fbIbBottleTransferAfterDragAfterSensor		(bIN:=
											P00_PackML.fbPMLAuto.ePMLState = E_PMLState.ePMLState_EXECUTE AND P13_BottleTransferAfterDrag.IbBottleTransferAfterDragAfterSensor													
											,tFilterTimeOn:=T#0MS, tFilterTimeOff:=T#500MS);
fbIbBottleTransferAfterDragSecondFormSensor		(bIN:=
											P00_PackML.fbPMLAuto.ePMLState = E_PMLState.ePMLState_EXECUTE AND P13_BottleTransferAfterDrag.IbBottleTransferAfterDragSecondFormSensor													
											,tFilterTimeOn:=T#35MS, tFilterTimeOff:=T#35MS);
rtfbIbBottleTransferAfterDragSecondFormSensor (CLK:=fbIbBottleTransferAfterDragSecondFormSensor.bOUT,Q=>);
IF rtfbIbBottleTransferAfterDragSecondFormSensor.Q THEN
	rtfbIbBottleTransferAfterDragSecondFormSensorCounter := rtfbIbBottleTransferAfterDragSecondFormSensorCounter + 1;
END_IF
tonrtfbIbBottleTransferAfterDragSecondFormSensorCounter(IN:=	rtfbIbBottleTransferAfterDragSecondFormSensorCounter<2 AND 
																P13_BottleTransferAfterDrag.IbBottleTransferAfterDragFirstFormSensor AND
																P13_BottleTransferAfterDrag.IbBottleTransferAfterDragSecondFormSensor AND
																bFormTransportersAfterScrewerCmdStart
														,PT := T#10S);
IF tonrtfbIbBottleTransferAfterDragSecondFormSensorCounter.Q THEN
	rtfbIbBottleTransferAfterDragSecondFormSensorCounter := 2;
END_IF

tonBottleTransferAfterDrag (IN:= 
								(P00_PackML.fbPMLAuto.ePMLState = E_PMLState.ePMLState_EXECUTE) AND 
								NOT (P00_PackML.fbPMLAuto.ePMLState = E_PMLState.ePMLState_STOPPING) AND
								P13_BottleTransferAfterDrag.fbBottleTransferAfterDrag.eState = E_Station.eReady AND 

								P13_BottleTransferAfterDrag.IbBottleTransferAfterDragFirstFormSensor AND
								rtfbIbBottleTransferAfterDragSecondFormSensorCounter >=2 
								//P13_BottleTransferAfterDrag.IbBottleTransferAfterDragSecondFormSensor,	
							,PT:=T#0MS);
P01_PucksInserter.IbPucksInserterFormGateAfterSensor;// Czujnik za PI						
						
IF tonBottleTransferAfterDrag.Q AND 
	NOT P13_BottleTransferAfterDrag.fbBottleTransferAfterDrag.bCycleDone AND
	NOT fbIbBottleTransferAfterDragAfterSensor.bOUT
THEN
	VIS.bBottleTransferAfterDragRun	:= TRUE;
END_IF

IF P13_BottleTransferAfterDrag.fbBottleTransferAfterDrag.bCycleDone THEN
	VIS.bBottleTransferAfterDragRun	:= FALSE;
	rtfbIbBottleTransferAfterDragSecondFormSensorCounter:= 0;
END_IF
END_ACTION

ACTION aP14_BadBottleConveyor:

(*************TRANSPORTER ODRZUCONYCH BUTELEK****************)
(************Przeniesiono wyzej*****************************)

(*Załączany w programie robota jak jest dorzut butelki i kasowany po 30 sekundach*)
IF bBadBottleConveyorEnable THEN
	;
ELSE
	bBadBottleConveyorStart				:=	FALSE;
	bBadBottleConveyorStartTriggerDelay	:=	FALSE;
END_IF

//Opóznienie załączania transporeta
IF bBadBottleConveyorStartTriggerDelay AND P13_BottleTransfer.fbBottleTransfer.eRunningState = eRejected THEN
	bBadBottleConveyorStartTrigger			:= TRUE;
	bBadBottleConveyorStartTriggerDelay		:=FALSE;
END_IF

//Sterowanie transporterem odrzuconych butelek
rtBadBottleConvoyerStart	(CLK:=	bBadBottleConveyorStartTrigger);
tofBadBottleConveyorStart	(IN:=	rtBadBottleConvoyerStart.Q ,	PT:=T#10S);

IF rtBadBottleConvoyerStart.Q THEN //Uruchamianie na cykl
	bBadBottleConveyorStartTrigger		:=	FALSE;
END_IF
IF NOT tofBadBottleConveyorStart.Q  THEN
	bBadBottleConveyorStart				:=	FALSE;
	bBadBottleConveyorStartTrigger		:=	FALSE;
ELSE
	bBadBottleConveyorStart 			:=	TRUE;	
END_IF
END_ACTION

ACTION aP15_FormTransporters:
(********Transporter przed dozownikami*************)
tofbFormTransportersDispencerSlow			(IN:=bFormTransportersDispencerSlowSpeedPulse, 	PT:=T#60S);
tonbFormTransportersDispencerResetSpeed		(IN:=bFormTransportersDispencerResetSpeed, 		PT:=T#5S);
tonQueBeforeScrewers						(IN:=P10_GripperScrewer.IbGripperScrewersSixthFormCheckFormSensor, PT:=T#1500mS);
tonQueAfterScrewers							(IN:=P11_CapCorrectCheck.IbCapCorrectCheckAfterScrewerFormSensor AND P11_CapCorrectCheck.IbCapCorrectCheckDialAfterScrewerFormSensor, PT:=T#2S);
tonQueAfterPlatin							(IN:=MAIN.IbLidSealerAfterSensor, PT:=T#3S);
tonQueBeforeDispencers						(IN:=MAIN.IbFormCheckFormSensor, PT:=T#2S);
tonDelayedStartAfterDisp					(IN:=NOT P09_CapPuttedCheck.fbIbCapPuttedCheckFormSensor.bOUT, PT:=T#1.5S);
IF GVL.bFormTransportersEnable AND (P00_PackML.fbPMLAuto.ePMLState = E_PMLState.ePMLState_EXECUTE)  THEN
	IF NOT VIS.bDosingTwoPhasesShow  THEN
		bFormTransportersDispencerCmdStart := TRUE;
	ELSIF VIS.bDosingTwoPhasesShow AND	NOT bFormTransportersScrewerStop AND NOT tonQueAfterPlatin.q THEN
		bFormTransportersDispencerCmdStart := TRUE;	
	END_IF
	bFormTransportersDispencerSlowSpeedPulse	:=	FALSE;
	(*Spowalnianie transportera*)	
	IF tofbFormTransportersDispencerSlow.Q AND NOT tonbFormTransportersDispencerResetSpeed.Q THEN
		bFormTransportersDispencerSlowSpeed	:= NOT VIS.bCapPuttedCheckIgnoreErrors; 
	ELSE
		bFormTransportersDispencerSlowSpeed	:= FALSE;
	END_IF
	IF bDosingTwoPhases THEN
		bFormTransportersDispencerSlowSpeed	:= TRUE;
	END_IF	
END_IF
	(*Wydmuch na tym transporterze*)
	QbBlowAfterGripperScrewer :=	bFormTransportersDispencerSlowSpeed;
(********Koniec Transporter przed dozownikami********)
	
(********Transporter za dozownikami*************)
tonbFormTransportersScrewerStop	(IN:=	(P05_Weight.eWeightStationRunningState = E_WeightLiftStationState.eStorageOfForms) AND 
										P05_Weight.fbWeightStation.iFormsCounterWeight1 >=3 AND 
										P05_Weight.fbWeightStation.iFormsCounterWeight2 >=3 AND 
										P05_Weight.fbWeightStation.iFormsCounterWeight3 >=3 AND 
										P05_Weight.fbWeightStation.iFormsCounterWeight4 >=3,
									PT:=T#500MS);
tofFormTransportersScrewerSlowSpeed	(IN:=P00_ReadRFIDCard.bReadedCardCapSorter AND bDosingTwoPhases, PT:=T#2S500MS);

IF 	P10_GripperScrewer.fbGripperScrewersDragStation.eRunningState = E_DragStationState.eEndingOfDrag  OR tonThirdFormCheckFormSensor.q THEN
//IF 	P10_GripperScrewer.fbGripperScrewersDragStation.eRunningState = E_DragStationState.eDraging AND P10_GripperScrewer.QbGripperScrewersDragLeadBefore1Actuator THEN
	bFormTransportersScrewerStop			:= FALSE;
END_IF


IF tonLongDelayAfterStart.Q AND
		eBeforeCapSorterPackageState[4].bFormPresent  AND
		(tonCapSorterFourthFormatSensorAnRegister.Q AND iCapSorterDragFormCounter >= 4)AND 
		MAIN.IbCapSorterBeforeFourthFormCheckFormSensor 
		THEN
			IF 
				NOT (
					(P05_Weight.eWeightStationRunningState = E_WeightLiftStationState.eStorageOfForms) AND 
					P05_Weight.fbWeightStation.iFormsCounterWeight1 =3 AND 
					P05_Weight.fbWeightStation.iFormsCounterWeight2 =3 AND 
					P05_Weight.fbWeightStation.iFormsCounterWeight3 =3 AND 
					P05_Weight.fbWeightStation.iFormsCounterWeight4 =3 
					)
				AND NOT bFormTransportersScrewerStop	
				//?AND NOT bLidFeederEnable
				(*AND NOT bDosingTwoPhases*)
				AND NOT bPhaseChanging
				AND tonDelayAfterStart.Q
				//AND (tonQueAfterScrewers.Q OR tonQueBeforeScrewers.Q)  //vs testy
			THEN
				bFormTransportersScrewerStop				:= 	TRUE;
			END_IF
		//bFormTransportersScrewerStop				:= 	TRUE;
END_IF
tonQueAfterScrewers.Q; tonQueBeforeScrewers.Q;
//IF bFormTransportersEnable AND (P00_PackML.fbPMLAuto.ePMLState = E_PMLState.ePMLState_EXECUTE)THEN //dp
IF bDelayAfterStart AND (*tonDelayAfterStart.Q AND*) bFormTransportersEnable AND (P00_PackML.fbPMLAuto.ePMLState = E_PMLState.ePMLState_EXECUTE OR 
		P00_PackML.fbPMLAuto.ePMLState = E_PMLState.ePMLState_STOPPING) (*AND tonDelayedStartAfterDisp.q co to*) THEN
	bFormTransportersScrewerCmdStart 			:= TRUE;
	tonbCapSorterOrCapSorterDragError.Q; 		//Spowalnianie transportera dla wag
	IF bFormTransportersScrewerStop	(*AND NOT tonbCapSorterOrCapSorterDragError.Q)*) THEN //Zatrzymywanie
		bFormTransportersScrewerCmdStart 		:= FALSE;
		
	END_IF
	//Vasyl na prośbę Karola
	(*IF (VIS.bDosingTwoPhasesShow OR vis.bLidFeederEnableShow) AND	tonQueAfterPlatin.Q OR bFormTransportersScrewerStop AND tonQueBeforeDispencers.q THEN
		bFormTransportersDispencerCmdStart 		:= FALSE;
	END_IF*)
END_IF

(********Transporter za sorterem nasadek*************)
IF bFormTransportersEnable AND (P00_PackML.fbPMLAuto.ePMLState = E_PMLState.ePMLState_EXECUTE)  THEN
	bFormTransportersAfterCapSorterCmdStart := TRUE;
	IF tonQueBeforeScrewers.Q THEN
		bFormTransportersAfterCapSorterCmdStart := FALSE;
	END_IF
END_IF	
	
(********Transporter przed zakręcarkami**************)
IF bFormTransportersEnable AND (P00_PackML.fbPMLAuto.ePMLState = E_PMLState.ePMLState_EXECUTE)  THEN
	bFormTransportersBeforeScrewerCmdStart := TRUE;
END_IF	

(*Wydmuch na tym transporterze*)
fbIbBlowBeforeGripperScrewerSensor		(bIn:=MAIN.IbBlowBeforeGripperScrewerSensor, tFilterTimeon:=T#5MS, tFilterTimeOff:=T#300MS);
fbIbBlowBeforeGripperScrewerSensor2		(bIn:=MAIN.IbBlowBeforeGripperScrewerSensor, tFilterTimeon:=T#100MS, tFilterTimeOff:=T#300MS);
tonBlowBeforeGripperScrewerSensor 		(IN:=MAIN.IbBlowBeforeGripperScrewerSensor, PT:=T#15S);
tpfbIbBlowBeforeGripperScrewerSensor 	(IN:=fbIbBlowBeforeGripperScrewerSensor.bOUT, PT:=T#1S);
QbBlowBeforeGripperScrewer	:=	fbIbBlowBeforeGripperScrewerSensor.bOut AND NOT tonBlowBeforeGripperScrewerSensor.Q;

(*Spowalniacz/szlabanik przed zakrecarkami*)
fbIbGateBeforeGripperScrewerSensor 		(bIn:=IbGateBeforeGripperScrewerSensor, tFilterTimeon:=T#20MS, tFilterTimeOff:=T#0MS);
fb2IbGateBeforeGripperScrewerSensor 	(bIn:=IbGateBeforeGripperScrewerSensor, tFilterTimeon:=T#400MS, tFilterTimeOff:=T#0MS);//bylo 670
ftfbIbGateBeforeGripperScrewerSensor	(CLK:=fbIbGateBeforeGripperScrewerSensor.bOUT,	Q=>);	
IF ftfbIbGateBeforeGripperScrewerSensor.Q THEN
	bGateBeforeGripperScrewer	:= TRUE;
END_IF
tonbGateBeforeGripperScrewer			(IN:=bGateBeforeGripperScrewer, PT:=T#400MS);
IF tonbGateBeforeGripperScrewer.Q THEN
	bGateBeforeGripperScrewer	:= FALSE;
END_IF
toniGateBeforeGripperScrewerCase1 (IN:=	iGateBeforeGripperScrewerCase = 10, PT:=T#4S);
						
CASE iGateBeforeGripperScrewerCase OF
	0:
		QbGateBeforeGripperScrewer 		:=	TRUE;
		iGateBeforeGripperScrewerCase	:=	iGateBeforeGripperScrewerCase	+	10;
	10:
		IF toniGateBeforeGripperScrewerCase1.Q AND NOT P09_CapPuttedCheck.IbCapPuttedCheckFormSensor THEN
			iGateBeforeGripperScrewerCase	:=	iGateBeforeGripperScrewerCase	+	10;
		END_IF
	20:
		QbGateBeforeGripperScrewer		:=	FALSE;
		iGateBeforeGripperScrewerCase	:=	iGateBeforeGripperScrewerCase	+	10;
	30: 
		QbGateBeforeGripperScrewer :=		fb2IbGateBeforeGripperScrewerSensor.bOUt;
END_CASE
	
//Spowalnianie formatek
iFormBeforeScrewers := 		
                       		BOOL_TO_INT(eBeforeScrewers2PackageState[2].bFormPresent)+
                       		BOOL_TO_INT(eBeforeScrewers2PackageState[1].bFormPresent)+
                       		BOOL_TO_INT(eBeforeScrewersPackageState[2].bFormPresent)+
                       		BOOL_TO_INT(eBeforeScrewersPackageState[1].bFormPresent);

tonCapPuttedFormsCheck			(IN:=	P10_GripperScrewer.IbGripperScrewersSixthFormCheckFormSensor,		PT:=T#80MS); //bylo 130
tonThirdFormCheckFormSensor		(IN:=	NOT P10_GripperScrewer.IbGripperScrewersSixthFormCheckFormSensor ,	PT:=T#30MS);
IF // Zatrzymywanie jeżeli
	tonCapPuttedFormsCheck.Q OR 			
	P00_PackML.fbPMLAuto.ePMLState = E_PMLState.ePMLState_STOPPING 	OR	
	NOT tonDelayAfterStart.Q	
THEN
	bFormTransporterSlowerCmdStart := FALSE;
END_IF
IF bDelayAfterStart AND bFormTransportersEnable AND 
	(
		tonThirdFormCheckFormSensor.Q OR 
		(NOT bDelayAfterStartFullRegister AND NOT P09_CapPuttedCheck.IbCapPuttedCheckFormSensor) OR
		(bDelayAfterStartFullRegister AND iFormBeforeScrewers=2) //do usuniecia
	)
	AND
	NOT (P00_PackML.fbPMLAuto.ePMLState = E_PMLState.ePMLState_STOPPING) 
	THEN 
		bFormTransporterSlowerCmdStart := TRUE;
END_IF

(********Transporter za zakręcarkami**************)
IF bFormTransportersEnable AND (P00_PackML.fbPMLAuto.ePMLState = E_PMLState.ePMLState_EXECUTE)  THEN
	bFormTransportersAfterScrewerCmdStart := TRUE;
END_IF
END_ACTION

ACTION aP16_LabelMachines:
(***********P16_LabelMachines**************)
(******************************************)
IF bLabelMachineEnable THEN
	bLabelMachineCmdStart := TRUE;
ELSE
	bLabelMachineCmdStart := FALSE;	
END_IF
(******************************************)
(******************************************)
END_ACTION

ACTION aP17_TurnTables:
(************P17_TurnTables****************)
(******************************************)

IF bExitTurnTableEnable AND bDelayAfterStart THEN
	bExitTurnTableCmdStart := TRUE;
ELSIF bDelayAfterStart THEN
	;//bExitTurnTableCmdStart := FALSE;
END_IF
(******************************************)
(******************************************)
IF bExitConveyorEnable AND bDelayAfterStart THEN
	bExitConveyorCmdStart := TRUE;
ELSE
	;//bExitConveyorCmdStart := FALSE;
END_IF
(******************************************)
(******************************************)


(*********************************************************)
(*********Szlaban na transporterze odbiorczym*************)
//Jeżeli stół pracuje 
bExitConveyorCmdStart;
//To ruszaj szlabanem
bExitConveyorGateRun;
//Czujnik z szlabanem
P17_TurnTables.IbExitConveyorGateAfterSensor;
P17_TurnTables.IbExitConveyorGateAfterSensor2;
IF bExitConveyorCmdStart THEN
	fbIbExitConveyorGateAfterSensor		(bIN:=P17_TurnTables.IbExitConveyorGateAfterSensor,	tFilterTimeOn:=T#10MS,	tFilterTimeOff:=T#10MS);
	fbIbExitConveyorGateAfterSensor2	(bIN:=P17_TurnTables.IbExitConveyorGateAfterSensor2,tFilterTimeOn:=T#1S800MS,	tFilterTimeOff:=T#1S800MS);
	tonbExitConveyorGateRun				(IN:=bExitConveyorGateRun AND NOT fbIbExitConveyorGateAfterSensor.bOUT, 	PT:=T#300MS);
	
	bExitConveyorGateRun S= fbIbExitConveyorGateAfterSensor.bOut;	
	bExitConveyorGateRun R= tonbExitConveyorGateRun.Q;	
	
	IF fbIbExitConveyorGateAfterSensor2.bOut AND bExitConveyorGateRun THEN
		bExitConveyorGateRunTemp := TRUE;
	ELSIF NOT fbIbExitConveyorGateAfterSensor2.bOut THEN
		bExitConveyorGateRunTemp := FALSE;	
	END_IF
	IF bExitConveyorGateRunTemp THEN
		bExitConveyorGateRun	:=	TRUE;
	END_IF
END_IF
(*********************************************************)
(*********************************************************)
	fbIbExitConveyorGateAfterSensor3		(bIN:=P17_TurnTables.IbExitConveyorGateAfterSensor,	tFilterTimeOn:=T#10MS,	tFilterTimeOff:=T#12S);

IF tonNotExecute.Q AND NOT fbIbExitConveyorGateAfterSensor3.bOut THEN
	bExitTurnTableCmdStart := FALSE;
	bExitConveyorCmdStart := FALSE;
END_IF
END_ACTION

END_PROGRAM

(* stored: Version 1.1.0.1, ProductVersion 3.1.4026.13, FileIdentifier 411a00112639a9e7228e2dd2d6e06ed5d9c97a99, FileSignature 68d56f6f7cd023b1b7825046622d1bf8a0b812843790b8bb4421e9821bde7a660f56d9956663ebebe51dd14dbbf8236e075714483451083181fa8ec4dce18396552c98323adbd34d97d4a2183e173e6a79f00ccb83a6e16e8aa8d04c780698a18ddc75a4fdb53c6e0a5ad36b78cb566d6a015d5d488b0f36d33e108bc6e3947adc481485b9a785ae4955bba34f0f1973acdd1e36ad2dc3e1a0f49b4145bd6d87dcf949c93894586451675c2a70766f69423c8f864f2bd740daf309413cd2660d30a041a2064fbf69f03032e63452ecfc9f4f022dbc58b6cc8660d268e867e61278df3a041a7dc567f471a15f51f76fbc6f01ffd4ca64c70a460cc0ac4c56d873
   POU P00_PackML: Id {bb851725-25aa-4e37-a964-31b2adf51159}, SpecialFunc None
   Folder CycleLogic: Id {06cd4f29-1d4a-4562-a5b5-d65a5d63923d}
   Folder Homing: Id {cd69f01d-dff3-44b8-b479-c86f6f37d13a}
   Folder Others: Id {4eaa7fda-3f18-47f1-b364-12a902042f69}
   Folder PML: Id {0da3c268-e19f-41cb-aa11-c303f93e5e7c}
   Folder PMLCommonStates: Id {650a41a5-55ef-4702-bbaa-88ebcf63e664}
   Action ACT_Aborted: Id {58aa837e-c8fc-4c28-9ce0-4a427a6cab20}
   Action ACT_Aborting: Id {6a678a84-5a61-4250-a4be-abf00b56123e}
   Action ACT_AntyError: Id {c7865532-fee1-4504-9555-bab70b080968}
   Action ACT_CapSorterBottleSorterAutoStart: Id {c3fb2df5-496e-4d6e-b52b-194c6aba5684}
   Action ACT_Clearing: Id {4fb303d6-b538-45f5-9c59-d20965484409}
   Action ACT_CycleLogic: Id {3da44b98-718e-4e63-9d16-900d089a9e0c}
   Action ACT_CycleLogicInIdle: Id {e572c3e4-a008-4c93-9a0f-a8917bea437f}
   Action ACT_CycleReset: Id {d01f058e-7391-4466-bfb0-8acae6a28ac8}
   Action ACT_CycleStarting: Id {bd94dca2-3142-49c3-b096-7cebb6d1d981}
   Action ACT_HandlingCommands: Id {112d64b6-2b07-417a-945d-df05a9d8b938}
   Action ACT_HomingCanceled: Id {c6fee273-32c9-4865-b5eb-8abdbdbe93ac}
   Action ACT_HomingCycle: Id {86cdacab-35ec-446f-bfbf-11166a6311e1}
   Action ACT_Mode: Id {fede3523-2f66-483b-a380-432be26a6954}
   Action ACT_ModeAutomatic: Id {60d63169-3a6d-4d59-8aa7-a7c32f5d2c01}
   Action ACT_ModeAutomaticConfectionEnding: Id {edf87eda-f614-4105-b905-991c76b97aa6}
   Action ACT_ModeManual: Id {0cdc2ae8-b7c4-4597-a9b1-f5a7c92f60e7}
   Action ACT_PhaseChanging: Id {49301ca2-85c3-4dbd-8b6d-5bd8ac1ba66f}
   Action ACT_PmlChangeMode: Id {34b871c7-b18a-4be6-8081-6f68dccece1a}
   Action ACT_PmlModeManager: Id {f475baa8-3f62-444c-a7ce-31090dd81ead}
   Action ACT_PmlResetCommands: Id {02e458fd-7054-41a9-a60e-5e60b9a76978}
   Action ACT_PmlStates: Id {d98c6e71-12ca-4dfc-b79f-6c185bff2953}
   Action ACT_PositioningLogic: Id {33c2de85-0726-4bc1-89a1-966bd1ecf91a}
   Action ACT_ResetAfterError: Id {384ae2de-ca7a-4fe1-9a03-166bdb49226d}
   Action ACT_ResetAfterErrorOrEstop_do_usun: Id {d5a90c27-226e-4f24-87ee-e7c3283c48e6}
   Action ACT_ResetAfterStart: Id {40d4e467-9ece-499e-a458-c346829ebf86}
   Action ACT_ResetCommands: Id {9ec0897e-36e7-4987-9141-27b6d559d720}
   Action ACT_ResetCommandsHoming: Id {aac1c86e-1a38-4119-b8ff-cf436b6068d8}
   Action ACT_Resetting: Id {060ba211-2928-4a5c-b275-16cea89f8390}
   Action ACT_SafetyFirstResetDelay: Id {e1cad260-5f2c-4b87-a53c-906e03b68232}
   Action ACT_Signals: Id {bf795528-045e-45d6-af15-735a7605ca13}
   Action ACT_SignalsFormsCounting: Id {4ecdb83e-025e-4855-82e6-aaf34a4915dc}
   Action ACT_SignalsLidFeeder: Id {ce6345bc-6574-4f36-9d19-cd1ab4c41b29}
   Action ACT_SignalsROPP: Id {c674e3d5-d02e-4129-a955-992ce939c175}
   Action ACT_Statistics: Id {d4fa1f1b-459a-48ee-ac8a-9a219e33f5f4}
   Action ACT_Stopped: Id {7f48db21-95cf-43c1-aeaf-872a57c426e9}
   Action ACT_Stopping: Id {ec11636e-9786-4f80-821f-df48323c100b}
   Action ACT_XtsChangeMode: Id {8d9ee5a4-afd7-49c1-82ef-d9259616fcb9}
   Action aP00_SingleRealeseIfNoCapBeforeScrewers: Id {03957123-98c2-4169-93f1-27c11007ade8}
   Action aP01_Barriers: Id {0504a637-224c-4002-9588-f2b1a391e77c}
   Action aP01_BottleFeeder: Id {a2cefbac-0c80-44a1-ad89-96d397551c5b}
   Action aP01_BottleSorter: Id {b0ffbba6-c622-483b-acc2-1cb969265347}
   Action aP01_Gates: Id {115f0cef-92dd-47a3-aa3b-1586c7b7646f}
   Action aP01_GatesLidFeederBarrier: Id {f6744a42-21b1-4004-b827-38a3de793ba7}
   Action aP01_PucksInserter: Id {bd3d0b67-5da0-4645-9f52-bc70293b0091}
   Action aP02_BottlePusher: Id {53df047e-5524-49fb-aa4d-2b526c372ee9}
   Action aP02_Dispencers1Phase: Id {c38bb36c-d7ed-4736-87d2-8cb357ebbc8b}
   Action aP02_Dispencers2Phase: Id {f66fa091-3e81-4119-adc1-a779143f6a02}
   Action aP02_Drag1Phase_GateAfter: Id {5ab0a412-c7cf-461d-8344-33a4f7597431}
   Action aP02_Drag2Phase_GateAfter: Id {b203ff93-24ed-49f7-8c5c-e06477228c4b}
   Action aP02_DragCheck: Id {6b178ed8-dc77-4895-9124-b77ce042043d}
   Action aP05_Weight: Id {20f67b79-09cd-4c2c-a8fa-2c696614797a}
   Action aP05_WeightBlock: Id {758885c2-2db2-4251-ac8c-281d03304e20}
   Action aP05_WeightGateBefore: Id {638dbe91-93c7-44e8-ab95-fab4ba8dd72c}
   Action aP06_LidFeeder: Id {c3553097-45da-4dc3-ae51-c8a00be7445b}
   Action aP06_LidPuttedCheck: Id {4b8a85fc-86e8-43df-a4f6-457edea15b2c}
   Action aP06_LidSealer: Id {82265ca1-1880-4053-8138-9bacc064142f}
   Action aP06_LidSealerDrag: Id {b4fa754d-d19a-49dd-ab8f-81f8f6ab4c07}
   Action aP06_LidSealerDrag2Phase: Id {2c031bdf-4776-42fe-8f46-43319ba98bb5}
   Action aP06_WickFeeder: Id {120d80de-ea52-47a5-81c6-2985da431f9a}
   Action aP07_CapPusher: Id {e44dc8ae-368b-4cdf-9c9b-84d7cc45b385}
   Action aP07_ROPP: Id {7366a79f-f958-416e-98f8-9cc43fc8283f}
   Action aP08_CapFeeder: Id {b15a201b-df30-4ce9-9964-09e3d9d4f554}
   Action aP08_CapSorter: Id {18384a5d-bc26-41c0-b703-4196e8582a43}
   Action aP08_CapSorterCycleTime: Id {4fc00516-5048-41b1-a7a3-9274ccfa916f}
   Action aP09_CapPuttedCheck: Id {16b52d53-72aa-4664-a8b0-f84cc64581c7}
   Action aP10_GripperScrewer: Id {80296e40-f3ca-4392-b247-f899a09e192e}
   Action aP10_GripperScrewerGate: Id {94311593-e7a4-4d5f-b136-569c7a039b11}
   Action aP11_CapCorrectCheck: Id {5cceb20f-bd8a-4828-9a03-9a0432d01651}
   Action aP13_BottleTransfer: Id {81197df5-2eac-40f1-87ef-efca6035df06}
   Action aP13_BottleTransferAfterDrag: Id {d7505347-e91c-460b-a7d9-b455e4e8388b}
   Action aP14_BadBottleConveyor: Id {007243bc-0599-4964-b19d-b00ca30742e2}
   Action aP15_FormTransporters: Id {fccee26e-e931-42d9-bf1d-a43138188e39}
   Action aP16_LabelMachines: Id {375ff8ee-ba3d-4f41-8c0b-c47d85ae0a81}
   Action aP17_TurnTables: Id {9bbd5e11-f096-4a47-aa50-07c433e18381} *)
